// {attribute 'hide_all_locals'}
FUNCTION_BLOCK INTERNAL FINAL FB_RepeatedStringMessageTests IMPLEMENTS I_Message
VAR_INPUT
END_VAR
VAR_OUTPUT
END_VAR

(*
syntax = "proto3";

message RepStringTest {
      repeated string RepStrings = 1 [
        (tchaxx.ext.v1.array_length) = 16,
        (tchaxx.ext.v1.max_string_len) = 32];
    }
*)

VAR
    fbMessageParser : FB_MessageParser(ipMessage:= THIS^);
    fbMessageWriter : FB_MessageWriter(ipMessage:= THIS^);
    aTmpBuffer      : ARRAY[0..Param_PB.cMaxCharacter] OF BYTE := [SIZEOF(aTmpBuffer)(16#FF)];
END_VAR

VAR
    aRepeatedStrings    : ARRAY [0..15] OF STRING(32);
    nField1Index        : UDINT; 
END_VAR

{warning 'Add method implementation '}
(* Calculates the size of this message in Protocol Buffer wire format, in bytes.*)
METHOD CalculateSize : UDINT
END_METHOD

(* Merges the data from the specified coded input stream with the current message.*)
METHOD MergeFrom : HRESULT
VAR_IN_OUT
	fbParseCtx : FB_ParseContext;
END_VAR
VAR
    nTag    : UDINT;
END_VAR
nField1Index := 0;

fbParseCtx.SetTempBuffer(anyBuffer:= THIS^.aTmpBuffer);

REPEAT   
MergeFrom := fbParseCtx.ReadTag(nTag=>nTag);
IF SUCCEEDED(MergeFrom) AND nTag = 0 THEN
    EXIT;
END_IF;

IF FAILED(MergeFrom) THEN
    MergeFrom := MergeFrom;
    RETURN;
END_IF

CASE nTag OF
    16#0A:         // repeated string (1)
       MergeFrom := fbParseCtx.ReadRepeatedFieldString(
                    anyArray:= F_ToAnyType(THIS^.aRepeatedStrings),
                    anyFirstElem:= F_ToAnyType(THIS^.aRepeatedStrings[0]),
                    nFieldIndex:= THIS^.nField1Index);
           
 
ELSE
    MergeFrom := fbParseCtx.SkipLastField();
END_CASE

UNTIL (FAILED(MergeFrom) OR nTag = 0)
END_REPEAT
END_METHOD

{warning 'Add property implementation'}
PROPERTY MessageValue : T_Any
GET
END_GET
END_PROPERTY

PROPERTY PUBLIC Parser : REFERENCE TO FB_MessageParser
GET
Parser REF= THIS^.fbMessageParser;
END_GET
END_PROPERTY

(* Writer for this message.*)
PROPERTY Writer : REFERENCE TO FB_MessageWriter
GET
Writer REF= THIS^.fbMessageWriter;
END_GET
END_PROPERTY

{warning 'Add method implementation '}
{attribute 'analysis' := '-33'}
(* Writes the data to the given coded output stream.*)
METHOD WriteTo : HRESULT
VAR_IN_OUT
	(* Coded output stream to write the data to. *)
	fbWriteCtx	: FB_WriteContext;
END_VAR
END_METHOD

END_FUNCTION_BLOCK

(* stored: Version 1.1.0.1
   POU FB_RepeatedStringMessageTests: Id {5ec75848-e7f7-4133-b1dd-36f6b0136090}, SpecialFunc None
   Method CalculateSize: Id {0452dc27-cdc5-4b88-8b67-f0ed717c838b}
   Method MergeFrom: Id {2889f9ff-159c-4b88-9bc6-f55d0596e20d}
   Property MessageValue: Id {67d823ce-54d1-458c-856d-92f9d16fbd70}
   Get Get: Id {d6e3df71-b25b-4a3d-9256-24349cc0e012}
   Property Parser: Id {9d9a84d5-eb4a-4abb-8518-acd3e8a5cac7}
   Get Get: Id {8c3c704e-b042-4bc4-ba1e-c6444118c347}
   Property Writer: Id {d5fd582d-7322-4920-9b8b-87fb7bbb2716}
   Get Get: Id {cbf982c5-cabe-4399-a0c6-1f25dd4bef63}
   Method WriteTo: Id {312eaa5a-dd8d-4886-9dde-bce1bb39e67b} *)
